FUNCTION_BLOCK LIMIT (* limiter *)
  (* Standard: 61131-3; Classification: standard selection function; Description: Copyright (c) 2011 TU Wien ACIN This program and the accompanying materials are made available under the terms of the Eclipse Public License 2.0 which is available at https://www.eclipse.org/legal/epl-2.0/ SPDX-License-Identifier: EPL-2.0 *)
  (* Version 1.0, 2011-06-21, Monika Wenger, TU Wien ACIN *)
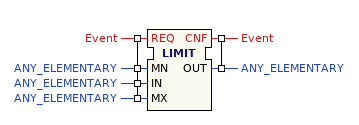
  EVENT_INPUT
    REQ WITH MN, MX, IN; (* Service Request *)
  END_EVENT
  EVENT_OUTPUT
    CNF WITH OUT; (* Confirmation of Requested Service *)
  END_EVENT
  VAR_INPUT
    MN : ANY_ELEMENTARY; (* Minimum *)
    IN : ANY_ELEMENTARY; (* Input *)
    MX : ANY_ELEMENTARY; (* Maximum *)
  END_VAR
  VAR_OUTPUT
    OUT : ANY_ELEMENTARY; (* Limited input *)
  END_VAR
END_FUNCTION_BLOCK
